PROGRAM Load_Mismatch_Active
VAR
END_VAR

Stationary.LoadMismatchCheckTrigger(CLK:= Stationary.LoadMismatchCheck, Q=> );

IF Stationary.LoadMismatchCheckTrigger.Q THEN
	
	//Told to pickup but have a load
	IF Otto.PickupLocation1 AND Stationary.LoadPresent[1] = FALSE THEN 
		
		Stationary.LoadMismatchActive	:= TRUE;
		
	ELSIF Otto.PickupLocation2 AND Stationary.LoadPresent[2] = FALSE THEN  
	
		Stationary.LoadMismatchActive	:= TRUE;
		
	ELSIF Otto.PickupLocation3 AND (Stationary.LoadPresent[1] = FALSE OR Stationary.LoadPresent[2] = FALSE) THEN 
		
		Stationary.LoadMismatchActive	:= TRUE;
		
	//Told to dropoff but are empty
	ELSIF Otto.DropoffLocation1 AND Stationary.LoadPresent[1] THEN 
		
		Stationary.LoadMismatchActive	:= TRUE;
		
	ELSIF Otto.DropoffLocation2 AND Stationary.LoadPresent[2] THEN  
	
		Stationary.LoadMismatchActive	:= TRUE;
		
	ELSIF Otto.DropoffLocation3 AND (Stationary.LoadPresent[1] OR Stationary.LoadPresent[2]) THEN 
		
		Stationary.LoadMismatchActive	:= TRUE;
		
	ELSE
		
		Stationary.LoadMismatchActive	:= FALSE;
		
	END_IF
	
END_IF

END_PROGRAM

(* stored: Version 1.1.0.1, ProductVersion 3.1.4024.9
   POU Load_Mismatch_Active: Id {39ae6742-6826-40b8-b67f-5ffed19e33b9}, SpecialFunc None *)
